// TIA Portal project "progettoPAGANOVOLZONE" (V17)
// Vorlageprojekt für das Buch mit Zielsystem S7-1200

(* hardware
DEVICE "S7-1200-Station_1"  S7-1200 Station
   slot 0: "Baugruppenträger_0"  Rack  V1.0
   slot 1: "PLC_1"  CPU 1215C DC/DC/DC  6ES7 215-1AG40-0XB0  V4.5
   slot 2: "DQ 2x24VDC _1"  SM 1222 DQ8 x 24VDC  6ES7 222-1BF30-0XB0  V1.0
DEVICE "HMI_1"  KTP900 Basic PN
   slot 0: "HMI_1"  KTP900 Basic PN  6AV2 123-2JB03-0AX0  17.0.0.0
   slot 1: "HMI_RT_1"  KTP900 Basic PN  6AV2 123-2JB03-0AX0  17.0.0.0
   slot 5: "HMI_1.IE_CP_1"  PROFINET Interface  17.0.0.0
      slot 1: "PROFINET Interface_1"  PROFINET Interface
         slot 1: "Port_1"  Port
*)

// ===== PLC "PLC_1"  CPU 1215C DC/DC/DC =====

VAR_GLOBAL   // PLC tag table "Standard-Variablentabelle"
   "Tag_1" AT %A0.0 : Bool;
   "Tag_2" AT %E0.0 : Bool;
   "Tag_3" AT %E0.1 : Bool;
   "Tag_4" AT %Q0.1 : Bool;
   "Tag_5" AT %I0.2 : Bool;
   "Tag_6" AT %Q0.2 : Bool;
   "Tag_7" AT %I0.3 : Bool;
   "Tag_8" AT %Q0.3 : Bool;
   "Tag_9" AT %I0.4 : Bool;
   "Tag_10" AT %Q0.4 : Bool;
   "Tag_11" AT %I0.5 : Bool;
   "Tag_12" AT %I0.6 : Bool;
   "Tag_13" AT %I0.7 : Bool;
   "Tag_14" AT %I1.0 : Bool;
   "Tag_15" AT %Q0.5 : Bool;
   "Tag_16" AT %Q0.6 : Bool;
   "Tag_17" AT %Q0.7 : Bool;
   "Tag_18" AT %Q1.0 : Bool;
   "Tag_19" AT %Q1.1 : Bool;
   "Tag_20" AT %I1.1 : Bool;
   "Tag_21" AT %I1.2 : Bool;
   "Tag_22" AT %Q1.2 : Bool;
   "Tag_23" AT %Q1.3 : Bool;
   "Tag_24" AT %I1.6 : Bool;
   "Tag_25" AT %ID30 : Real;
   "Tag_26" AT %I1.3 : Bool;
   "Tag_27" AT %I1.5 : Bool;
   "Tag_28" AT %I1.7 : Bool;
   "Tag_29" AT %Q1.4 : Bool;
   "Tag_30" AT %Q1.5 : Bool;
   "Tag_31" AT %Q1.6 : Bool;
   "Tag_32" AT %Q1.7 : Bool;
   "Tag_33" AT %I1.4 : Bool;
   "tag1" AT %M1.0 : Bool;
   "pezzi_scartati" AT %MW0 : Int;
   "allarme" AT %Q2.0 : Bool;
   "Tag_34" AT %I2.1 : Bool;
   "Tag_35" AT %I2.0 : Bool;
   "Tag_36" AT %I2.2 : Bool;
   "Tag_37" AT %I2.3 : Bool;
END_VAR

DATA_BLOCK "nastro1"   // DB1
{ S7_Optimized_Access := 'TRUE' }
VERSION : 0.1
// stored: InstanceOfName nastro
"nastro"
BEGIN
END_DATA_BLOCK

DATA_BLOCK "nastro2"   // DB2
{ S7_Optimized_Access := 'TRUE' }
VERSION : 0.1
// stored: InstanceOfName nastro
"nastro"
BEGIN
END_DATA_BLOCK

DATA_BLOCK "nastro3"   // DB3
{ S7_Optimized_Access := 'TRUE' }
VERSION : 0.1
// stored: InstanceOfName nastro
"nastro"
BEGIN
END_DATA_BLOCK

DATA_BLOCK "robotCentrale"   // DB5
{ S7_Optimized_Access := 'TRUE' }
VERSION : 0.1
// stored: InstanceOfName robotSD
"robotSD"
BEGIN
END_DATA_BLOCK

DATA_BLOCK "elevator1"   // DB7
{ S7_Optimized_Access := 'TRUE' }
VERSION : 0.1
// stored: InstanceOfName elevator
"elevator"
BEGIN
END_DATA_BLOCK

DATA_BLOCK "nastroCentrale1"   // DB8
{ S7_Optimized_Access := 'TRUE' }
VERSION : 0.1
// stored: InstanceOfName nastroCentrale
"nastroCentrale"
BEGIN
END_DATA_BLOCK

DATA_BLOCK "weight1"   // DB9
{ S7_Optimized_Access := 'TRUE' }
VERSION : 0.1
// stored: InstanceOfName weight
"weight"
BEGIN
END_DATA_BLOCK

DATA_BLOCK "NastroDirezionale1"   // DB10
{ S7_Optimized_Access := 'TRUE' }
VERSION : 0.1
// stored: InstanceOfName NastroDirezionale
"NastroDirezionale"
BEGIN
END_DATA_BLOCK

FUNCTION_BLOCK "robotSD"   // FB1, LAD
{ S7_Optimized_Access := 'TRUE' }
VERSION : 0.1
   VAR_INPUT
      workD : Bool;   // work del nastro destro
      workS : Bool;   // work del nastro sinistro
      grabsens : Bool;
      godownsens : Bool;
      movesens : Bool;
      rotateSens : Bool;
      occupato : Bool;   // sensore sul nastro d'arrivo
      tempot2 : Time := T#1s;
   END_VAR
   VAR_OUTPUT
      godown : Bool;
      grab : Bool;
      move : Bool;
      sinistra : Bool;
      destra : Bool;
      work_finishedD : Bool;
      work_finishedS : Bool;
   END_VAR
   VAR
      f0 : Bool;   // base
      "f1.1" : Bool;
      "f1.2" : Bool;
      f2 : Bool;
      f3 : Bool;
      f4 : Bool;
      "f5.1" : Bool;
      "f5.2" : Bool;
      f6 : Bool;
      f7 : Bool;
      f8 : Bool;
      f9 : Bool;
      "f9.1" : Bool;
      f10 : Bool;
      iniz : Bool;
      F_sensD : F_TRIG;   // falling del sensore destro
      F_sensS : F_TRIG;   // falling del sensore sinistro
      R_grabsens : R_TRIG;
      R_occupato : R_TRIG;
      F_godownsens : F_TRIG;
      F_movesens : F_TRIG;
      F_rotateSens : F_TRIG;   // falling del sensore di rotazione
      timer_f2 : TON_TIME;
      varDestra : Bool;
   END_VAR
   VAR_TEMP
      tr1 : Bool;   // sensore destro o sinistro falling edge
      tr2 : Bool;
      tr3 : Bool;
      tr4 : Bool;
      tr5 : Bool;
      tr6 : Bool;
      tr7 : Bool;
      tr8 : Bool;
      tr9 : Bool;
      tr10 : Bool;
      tr11 : Bool;
      tr12 : Bool;
      tr13 : Bool;
      tr14 : Bool;
      "tr14.1" : Bool;
      tr15 : Bool;
   END_VAR
   VAR_TEMP   // added for the SCL form of the ladder/FBD networks
      _w1 : Bool;
   END_VAR
BEGIN

REGION Network 1: inizializzazione
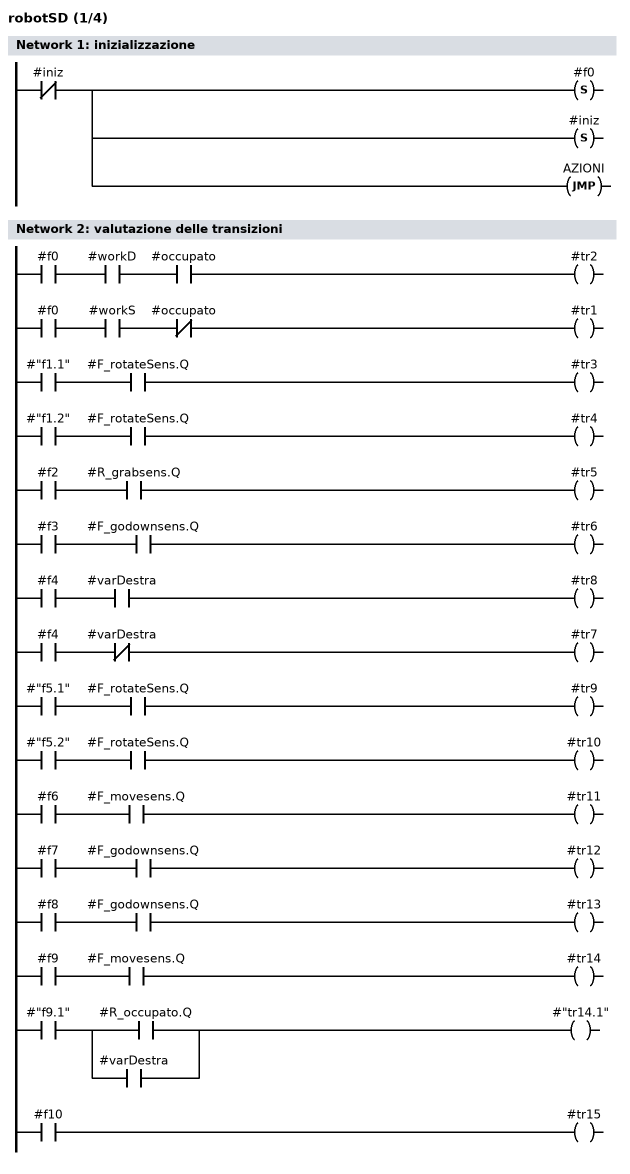
   RUNG wire#powerrail
      I_Contact( #iniz )
      wire#w1
      S_Coil( #f0 )
   END_RUNG
   RUNG wire#w1
      S_Coil( #iniz )
   END_RUNG
   RUNG wire#w1
      JumpCoil( AZIONI )
   END_RUNG
   // the same network as SCL:
   IF NOT #iniz THEN #f0 := TRUE; END_IF;
   #_w1 := NOT #iniz;
   IF #_w1 THEN
       #iniz := TRUE;
       GOTO AZIONI;
   END_IF;
END_REGION

REGION Network 2: valutazione delle transizioni
   RUNG wire#powerrail
      Contact( #f0 )
      Contact( #workD )
      Contact( #occupato )
      Coil( #tr2 )
   END_RUNG
   RUNG wire#powerrail
      Contact( #f0 )
      Contact( #workS )
      I_Contact( #occupato )
      Coil( #tr1 )
   END_RUNG
   RUNG wire#powerrail
      Contact( #"f1.1" )
      Contact( #F_rotateSens.Q )
      Coil( #tr3 )
   END_RUNG
   RUNG wire#powerrail
      Contact( #"f1.2" )
      Contact( #F_rotateSens.Q )
      Coil( #tr4 )
   END_RUNG
   RUNG wire#powerrail
      Contact( #f2 )
      Contact( #R_grabsens.Q )
      Coil( #tr5 )
   END_RUNG
   RUNG wire#powerrail
      Contact( #f3 )
      Contact( #F_godownsens.Q )
      Coil( #tr6 )
   END_RUNG
   RUNG wire#powerrail
      Contact( #f4 )
      Contact( #varDestra )
      Coil( #tr8 )
   END_RUNG
   RUNG wire#powerrail
      Contact( #f4 )
      I_Contact( #varDestra )
      Coil( #tr7 )
   END_RUNG
   RUNG wire#powerrail
      Contact( #"f5.1" )
      Contact( #F_rotateSens.Q )
      Coil( #tr9 )
   END_RUNG
   RUNG wire#powerrail
      Contact( #"f5.2" )
      Contact( #F_rotateSens.Q )
      Coil( #tr10 )
   END_RUNG
   RUNG wire#powerrail
      Contact( #f6 )
      Contact( #F_movesens.Q )
      Coil( #tr11 )
   END_RUNG
   RUNG wire#powerrail
      Contact( #f7 )
      Contact( #F_godownsens.Q )
      Coil( #tr12 )
   END_RUNG
   RUNG wire#powerrail
      Contact( #f8 )
      Contact( #F_godownsens.Q )
      Coil( #tr13 )
   END_RUNG
   RUNG wire#powerrail
      Contact( #f9 )
      Contact( #F_movesens.Q )
      Coil( #tr14 )
   END_RUNG
   RUNG wire#powerrail
      Contact( #"f9.1" )
      wire#w1
      Contact( #R_occupato.Q )
      wire#w2
      Coil( #"tr14.1" )
   END_RUNG
   RUNG wire#w1
      Contact( #varDestra )
   END_RUNG wire#w2
   RUNG wire#powerrail
      Contact( #f10 )
      Coil( #tr15 )
   END_RUNG
   // the same network as SCL:
   #tr2 := #f0 AND #workD AND #occupato;
   #tr1 := #f0 AND #workS AND NOT #occupato;
   #tr3 := #"f1.1" AND #F_rotateSens.Q;
   #tr4 := #"f1.2" AND #F_rotateSens.Q;
   #tr5 := #f2 AND #R_grabsens.Q;
   #tr6 := #f3 AND #F_godownsens.Q;
   #tr8 := #f4 AND #varDestra;
   #tr7 := #f4 AND NOT #varDestra;
   #tr9 := #"f5.1" AND #F_rotateSens.Q;
   #tr10 := #"f5.2" AND #F_rotateSens.Q;
   #tr11 := #f6 AND #F_movesens.Q;
   #tr12 := #f7 AND #F_godownsens.Q;
   #tr13 := #f8 AND #F_godownsens.Q;
   #tr14 := #f9 AND #F_movesens.Q;
   #"tr14.1" := #"f9.1" AND (#R_occupato.Q OR #varDestra);
   #tr15 := #f10;
END_REGION

REGION Network 3: aggiornamento della condizione
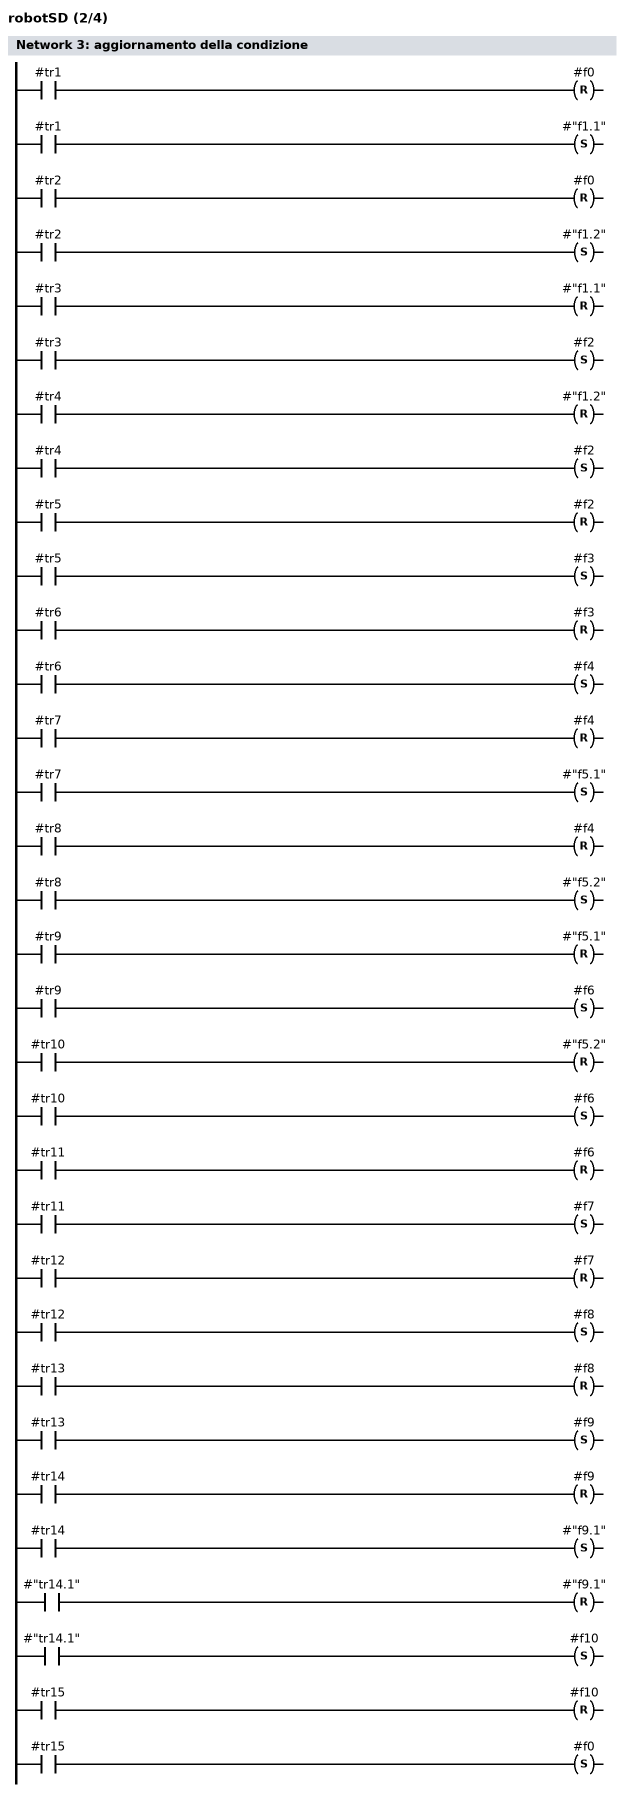
   RUNG wire#powerrail
      Contact( #tr1 )
      R_Coil( #f0 )
   END_RUNG
   RUNG wire#powerrail
      Contact( #tr1 )
      S_Coil( #"f1.1" )
   END_RUNG
   RUNG wire#powerrail
      Contact( #tr2 )
      R_Coil( #f0 )
   END_RUNG
   RUNG wire#powerrail
      Contact( #tr2 )
      S_Coil( #"f1.2" )
   END_RUNG
   RUNG wire#powerrail
      Contact( #tr3 )
      R_Coil( #"f1.1" )
   END_RUNG
   RUNG wire#powerrail
      Contact( #tr3 )
      S_Coil( #f2 )
   END_RUNG
   RUNG wire#powerrail
      Contact( #tr4 )
      R_Coil( #"f1.2" )
   END_RUNG
   RUNG wire#powerrail
      Contact( #tr4 )
      S_Coil( #f2 )
   END_RUNG
   RUNG wire#powerrail
      Contact( #tr5 )
      R_Coil( #f2 )
   END_RUNG
   RUNG wire#powerrail
      Contact( #tr5 )
      S_Coil( #f3 )
   END_RUNG
   RUNG wire#powerrail
      Contact( #tr6 )
      R_Coil( #f3 )
   END_RUNG
   RUNG wire#powerrail
      Contact( #tr6 )
      S_Coil( #f4 )
   END_RUNG
   RUNG wire#powerrail
      Contact( #tr7 )
      R_Coil( #f4 )
   END_RUNG
   RUNG wire#powerrail
      Contact( #tr7 )
      S_Coil( #"f5.1" )
   END_RUNG
   RUNG wire#powerrail
      Contact( #tr8 )
      R_Coil( #f4 )
   END_RUNG
   RUNG wire#powerrail
      Contact( #tr8 )
      S_Coil( #"f5.2" )
   END_RUNG
   RUNG wire#powerrail
      Contact( #tr9 )
      R_Coil( #"f5.1" )
   END_RUNG
   RUNG wire#powerrail
      Contact( #tr9 )
      S_Coil( #f6 )
   END_RUNG
   RUNG wire#powerrail
      Contact( #tr10 )
      R_Coil( #"f5.2" )
   END_RUNG
   RUNG wire#powerrail
      Contact( #tr10 )
      S_Coil( #f6 )
   END_RUNG
   RUNG wire#powerrail
      Contact( #tr11 )
      R_Coil( #f6 )
   END_RUNG
   RUNG wire#powerrail
      Contact( #tr11 )
      S_Coil( #f7 )
   END_RUNG
   RUNG wire#powerrail
      Contact( #tr12 )
      R_Coil( #f7 )
   END_RUNG
   RUNG wire#powerrail
      Contact( #tr12 )
      S_Coil( #f8 )
   END_RUNG
   RUNG wire#powerrail
      Contact( #tr13 )
      R_Coil( #f8 )
   END_RUNG
   RUNG wire#powerrail
      Contact( #tr13 )
      S_Coil( #f9 )
   END_RUNG
   RUNG wire#powerrail
      Contact( #tr14 )
      R_Coil( #f9 )
   END_RUNG
   RUNG wire#powerrail
      Contact( #tr14 )
      S_Coil( #"f9.1" )
   END_RUNG
   RUNG wire#powerrail
      Contact( #"tr14.1" )
      R_Coil( #"f9.1" )
   END_RUNG
   RUNG wire#powerrail
      Contact( #"tr14.1" )
      S_Coil( #f10 )
   END_RUNG
   RUNG wire#powerrail
      Contact( #tr15 )
      R_Coil( #f10 )
   END_RUNG
   RUNG wire#powerrail
      Contact( #tr15 )
      S_Coil( #f0 )
   END_RUNG
   // the same network as SCL:
   IF #tr1 THEN
       #f0 := FALSE;
       #"f1.1" := TRUE;
   END_IF;
   IF #tr2 THEN
       #f0 := FALSE;
       #"f1.2" := TRUE;
   END_IF;
   IF #tr3 THEN
       #"f1.1" := FALSE;
       #f2 := TRUE;
   END_IF;
   IF #tr4 THEN
       #"f1.2" := FALSE;
       #f2 := TRUE;
   END_IF;
   IF #tr5 THEN
       #f2 := FALSE;
       #f3 := TRUE;
   END_IF;
   IF #tr6 THEN
       #f3 := FALSE;
       #f4 := TRUE;
   END_IF;
   IF #tr7 THEN
       #f4 := FALSE;
       #"f5.1" := TRUE;
   END_IF;
   IF #tr8 THEN
       #f4 := FALSE;
       #"f5.2" := TRUE;
   END_IF;
   IF #tr9 THEN
       #"f5.1" := FALSE;
       #f6 := TRUE;
   END_IF;
   IF #tr10 THEN
       #"f5.2" := FALSE;
       #f6 := TRUE;
   END_IF;
   IF #tr11 THEN
       #f6 := FALSE;
       #f7 := TRUE;
   END_IF;
   IF #tr12 THEN
       #f7 := FALSE;
       #f8 := TRUE;
   END_IF;
   IF #tr13 THEN
       #f8 := FALSE;
       #f9 := TRUE;
   END_IF;
   IF #tr14 THEN
       #f9 := FALSE;
       #"f9.1" := TRUE;
   END_IF;
   IF #"tr14.1" THEN
       #"f9.1" := FALSE;
       #f10 := TRUE;
   END_IF;
   IF #tr15 THEN
       #f10 := FALSE;
       #f0 := TRUE;
   END_IF;
END_REGION

REGION Network 4: esecuzione delle azioni
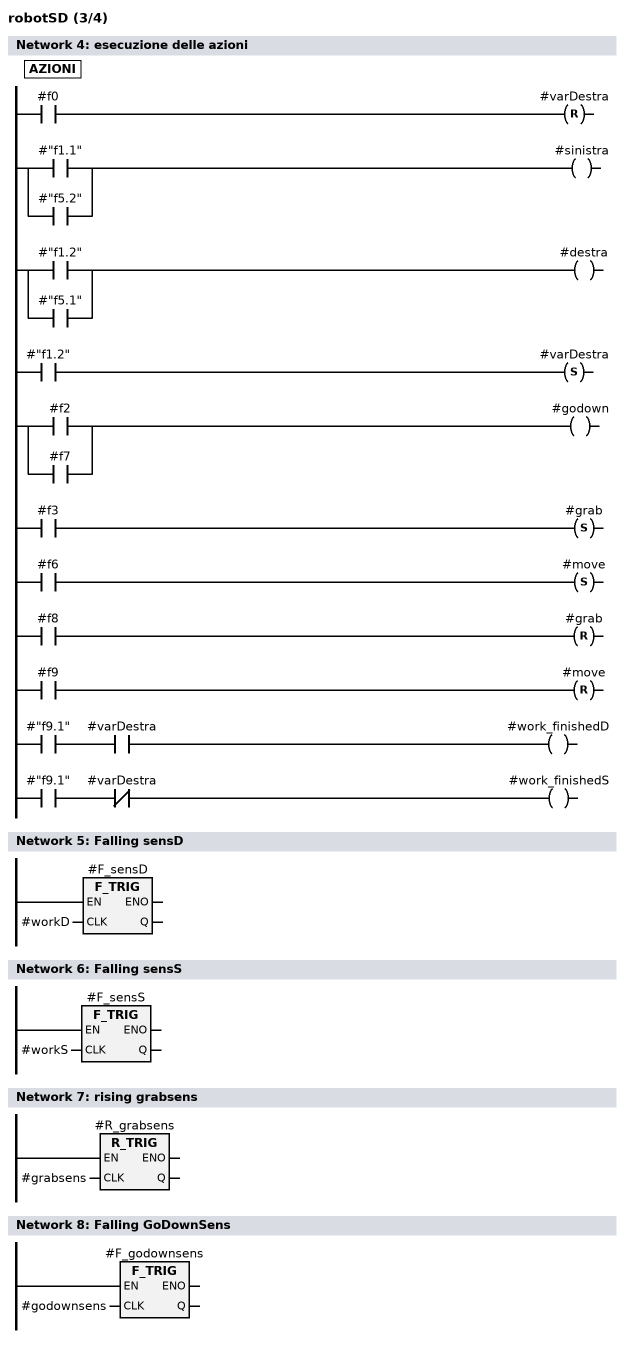
   Label( AZIONI )
   RUNG wire#powerrail
      Contact( #f0 )
      R_Coil( #varDestra )
   END_RUNG
   RUNG wire#powerrail
      Contact( #"f1.1" )
      wire#w1
      Coil( #sinistra )
   END_RUNG
   RUNG wire#powerrail
      Contact( #"f5.2" )
   END_RUNG wire#w1
   RUNG wire#powerrail
      Contact( #"f1.2" )
      wire#w2
      Coil( #destra )
   END_RUNG
   RUNG wire#powerrail
      Contact( #"f5.1" )
   END_RUNG wire#w2
   RUNG wire#powerrail
      Contact( #"f1.2" )
      S_Coil( #varDestra )
   END_RUNG
   RUNG wire#powerrail
      Contact( #f2 )
      wire#w3
      Coil( #godown )
   END_RUNG
   RUNG wire#powerrail
      Contact( #f7 )
   END_RUNG wire#w3
   RUNG wire#powerrail
      Contact( #f3 )
      S_Coil( #grab )
   END_RUNG
   RUNG wire#powerrail
      Contact( #f6 )
      S_Coil( #move )
   END_RUNG
   RUNG wire#powerrail
      Contact( #f8 )
      R_Coil( #grab )
   END_RUNG
   RUNG wire#powerrail
      Contact( #f9 )
      R_Coil( #move )
   END_RUNG
   RUNG wire#powerrail
      Contact( #"f9.1" )
      Contact( #varDestra )
      Coil( #work_finishedD )
   END_RUNG
   RUNG wire#powerrail
      Contact( #"f9.1" )
      I_Contact( #varDestra )
      Coil( #work_finishedS )
   END_RUNG
   // the same network as SCL:
   AZIONI:
   IF #f0 THEN #varDestra := FALSE; END_IF;
   #sinistra := #"f1.1" OR #"f5.2";
   #destra := #"f1.2" OR #"f5.1";
   IF #"f1.2" THEN #varDestra := TRUE; END_IF;
   #godown := #f2 OR #f7;
   IF #f3 THEN #grab := TRUE; END_IF;
   IF #f6 THEN #move := TRUE; END_IF;
   IF #f8 THEN #grab := FALSE; END_IF;
   IF #f9 THEN #move := FALSE; END_IF;
   #work_finishedD := #"f9.1" AND #varDestra;
   #work_finishedS := #"f9.1" AND NOT #varDestra;
END_REGION

REGION Network 5: Falling sensD
   #F_sensD(CLK := #workD);   // F_TRIG
END_REGION

REGION Network 6: Falling sensS
   #F_sensS(CLK := #workS);   // F_TRIG
END_REGION

REGION Network 7: rising grabsens
   #R_grabsens(CLK := #grabsens);   // R_TRIG
END_REGION

REGION Network 8: Falling GoDownSens
   #F_godownsens(CLK := #godownsens);   // F_TRIG
END_REGION

REGION Network 9: Falling MoveSens
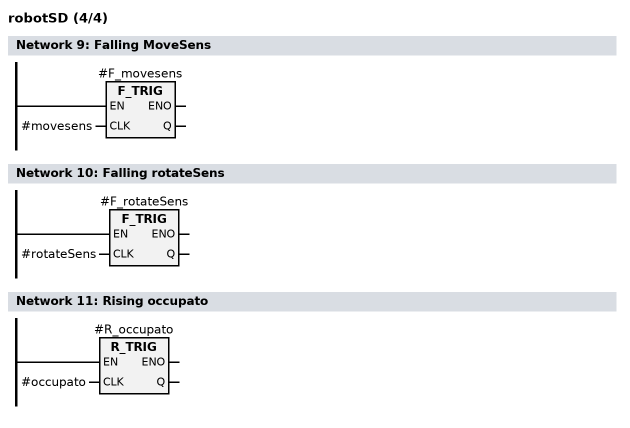
   #F_movesens(CLK := #movesens);   // F_TRIG
END_REGION

REGION Network 10: Falling rotateSens
   #F_rotateSens(CLK := #rotateSens);   // F_TRIG
END_REGION

REGION Network 11: Rising occupato
   #R_occupato(CLK := #occupato);   // R_TRIG
END_REGION
END_FUNCTION_BLOCK

FUNCTION_BLOCK "nastro"   // FB2, LAD
{ S7_Optimized_Access := 'TRUE' }
VERSION : 0.1
   VAR_INPUT
      s : Bool;
      work_finished : Bool;
   END_VAR
   VAR_OUTPUT
      motor : Bool;
      work : Bool;
   END_VAR
   VAR
      f0 : Bool;
      f1 : Bool;
      f2 : Bool;
      init : Bool;
      F_S : F_TRIG;
      F_Finished : F_TRIG;
      R_S : R_TRIG;
   END_VAR
   VAR_TEMP
      tr1 : Bool;
      tr3 : Bool;
      tr2 : Bool;
   END_VAR
   VAR_TEMP   // added for the SCL form of the ladder/FBD networks
      _w1 : Bool;
   END_VAR
BEGIN

REGION Network 1: inizializzazione
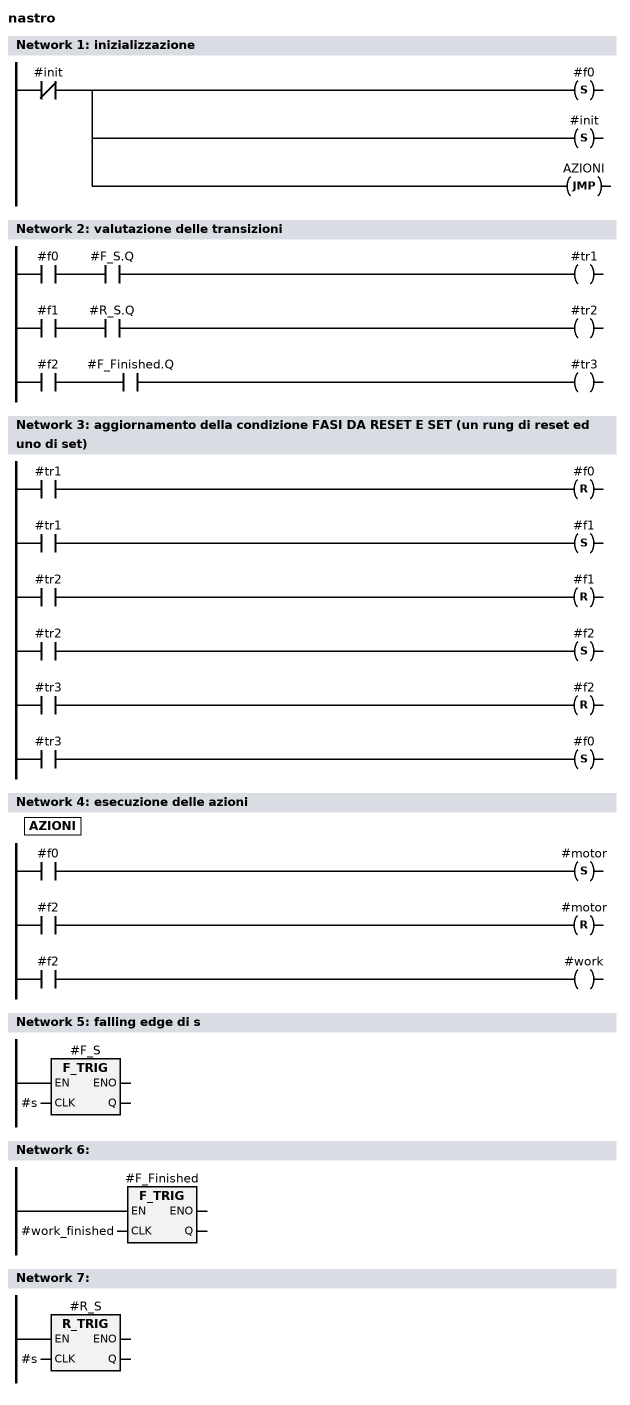
   RUNG wire#powerrail
      I_Contact( #init )
      wire#w1
      S_Coil( #f0 )
   END_RUNG
   RUNG wire#w1
      S_Coil( #init )
   END_RUNG
   RUNG wire#w1
      JumpCoil( AZIONI )
   END_RUNG
   // the same network as SCL:
   IF NOT #init THEN #f0 := TRUE; END_IF;
   #_w1 := NOT #init;
   IF #_w1 THEN
       #init := TRUE;
       GOTO AZIONI;
   END_IF;
END_REGION

REGION Network 2: valutazione delle transizioni
   RUNG wire#powerrail
      Contact( #f0 )
      Contact( #F_S.Q )
      Coil( #tr1 )
   END_RUNG
   RUNG wire#powerrail
      Contact( #f1 )
      Contact( #R_S.Q )
      Coil( #tr2 )
   END_RUNG
   RUNG wire#powerrail
      Contact( #f2 )
      Contact( #F_Finished.Q )
      Coil( #tr3 )
   END_RUNG
   // the same network as SCL:
   #tr1 := #f0 AND #F_S.Q;
   #tr2 := #f1 AND #R_S.Q;
   #tr3 := #f2 AND #F_Finished.Q;
END_REGION

REGION Network 3: aggiornamento della condizione FASI DA RESET E SET (un rung di reset ed uno di set)
   RUNG wire#powerrail
      Contact( #tr1 )
      R_Coil( #f0 )
   END_RUNG
   RUNG wire#powerrail
      Contact( #tr1 )
      S_Coil( #f1 )
   END_RUNG
   RUNG wire#powerrail
      Contact( #tr2 )
      R_Coil( #f1 )
   END_RUNG
   RUNG wire#powerrail
      Contact( #tr2 )
      S_Coil( #f2 )
   END_RUNG
   RUNG wire#powerrail
      Contact( #tr3 )
      R_Coil( #f2 )
   END_RUNG
   RUNG wire#powerrail
      Contact( #tr3 )
      S_Coil( #f0 )
   END_RUNG
   // the same network as SCL:
   IF #tr1 THEN
       #f0 := FALSE;
       #f1 := TRUE;
   END_IF;
   IF #tr2 THEN
       #f1 := FALSE;
       #f2 := TRUE;
   END_IF;
   IF #tr3 THEN
       #f2 := FALSE;
       #f0 := TRUE;
   END_IF;
END_REGION

REGION Network 4: esecuzione delle azioni
   Label( AZIONI )
   RUNG wire#powerrail
      Contact( #f0 )
      S_Coil( #motor )
   END_RUNG
   RUNG wire#powerrail
      Contact( #f2 )
      R_Coil( #motor )
   END_RUNG
   RUNG wire#powerrail
      Contact( #f2 )
      Coil( #work )
   END_RUNG
   // the same network as SCL:
   AZIONI:
   IF #f0 THEN #motor := TRUE; END_IF;
   IF #f2 THEN #motor := FALSE; END_IF;
   #work := #f2;
END_REGION

REGION Network 5: falling edge di s
   #F_S(CLK := #s);   // F_TRIG
END_REGION

REGION Network 6
   #F_Finished(CLK := #work_finished);   // F_TRIG
END_REGION

REGION Network 7
   #R_S(CLK := #s);   // R_TRIG
END_REGION
END_FUNCTION_BLOCK

FUNCTION_BLOCK "elevator"   // FB3, LAD
TITLE = elevatore
{ S7_Optimized_Access := 'TRUE' }
VERSION : 0.1
   VAR_INPUT
      piano : Bool;
      sensDXup : Bool;
      boxon : Bool;
      sensSTOP : Bool;
      elevatorDown : Bool;
      sensDXdown : Bool;
      sensS : Bool;
   END_VAR
   VAR_OUTPUT
      down : Bool;
      AVA : Bool;
      up : Bool;
      work_finished : Bool;
   END_VAR
   VAR
      f0 : Bool;   // work finished
      "f0.1" : Bool;
      "f1.1" : Bool;   // piano 1
      "f1.2" : Bool;   // piano 0
      "f2.1" : Bool;   // sopra
      "f3.1" : Bool;   // piano 1, scendere fino a piano 0
      f4 : Bool;
      init : Bool;
      F_sensDXup : F_TRIG;
      F_boxOn : F_TRIG;
      F_sensDXdown : F_TRIG;
      F_sensS : F_TRIG;
      R_sensStop : R_TRIG;
      R_elevatorDown : R_TRIG;
   END_VAR
   VAR_TEMP
      tr1 : Bool;
      tr2 : Bool;
      tr3 : Bool;
      "tr3.1" : Bool;
      tr4 : Bool;
      tr5 : Bool;
      tr6 : Bool;
      tr7 : Bool;
      "tr0.1" : Bool;
   END_VAR
   VAR_TEMP   // added for the SCL form of the ladder/FBD networks
      _w1 : Bool;
   END_VAR
BEGIN

REGION Network 1: inizializzazione
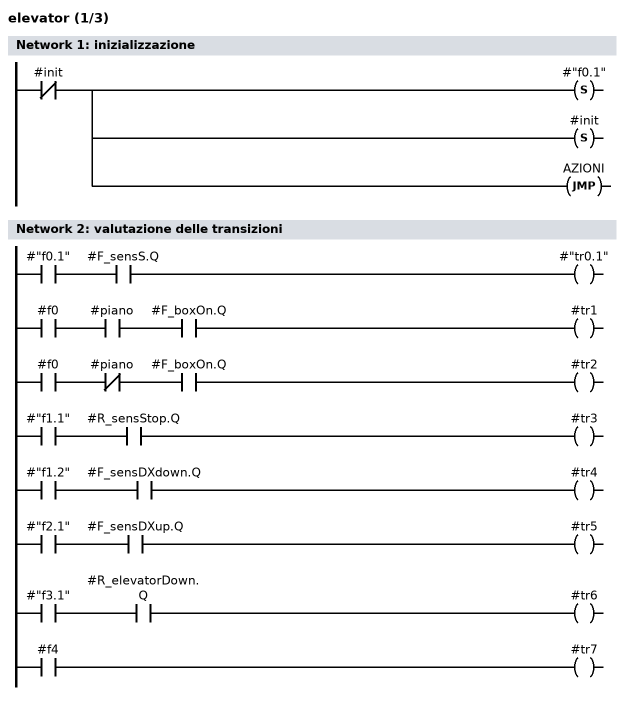
   RUNG wire#powerrail
      I_Contact( #init )
      wire#w1
      S_Coil( #"f0.1" )
   END_RUNG
   RUNG wire#w1
      S_Coil( #init )
   END_RUNG
   RUNG wire#w1
      JumpCoil( AZIONI )
   END_RUNG
   // the same network as SCL:
   IF NOT #init THEN #"f0.1" := TRUE; END_IF;
   #_w1 := NOT #init;
   IF #_w1 THEN
       #init := TRUE;
       GOTO AZIONI;
   END_IF;
END_REGION

REGION Network 2: valutazione delle transizioni
   RUNG wire#powerrail
      Contact( #"f0.1" )
      Contact( #F_sensS.Q )
      Coil( #"tr0.1" )
   END_RUNG
   RUNG wire#powerrail
      Contact( #f0 )
      Contact( #piano )
      Contact( #F_boxOn.Q )
      Coil( #tr1 )
   END_RUNG
   RUNG wire#powerrail
      Contact( #f0 )
      I_Contact( #piano )
      Contact( #F_boxOn.Q )
      Coil( #tr2 )
   END_RUNG
   RUNG wire#powerrail
      Contact( #"f1.1" )
      Contact( #R_sensStop.Q )
      Coil( #tr3 )
   END_RUNG
   RUNG wire#powerrail
      Contact( #"f1.2" )
      Contact( #F_sensDXdown.Q )
      Coil( #tr4 )
   END_RUNG
   RUNG wire#powerrail
      Contact( #"f2.1" )
      Contact( #F_sensDXup.Q )
      Coil( #tr5 )
   END_RUNG
   RUNG wire#powerrail
      Contact( #"f3.1" )
      Contact( #R_elevatorDown.Q )
      Coil( #tr6 )
   END_RUNG
   RUNG wire#powerrail
      Contact( #f4 )
      Coil( #tr7 )
   END_RUNG
   // the same network as SCL:
   #"tr0.1" := #"f0.1" AND #F_sensS.Q;
   #tr1 := #f0 AND #piano AND #F_boxOn.Q;
   #tr2 := #f0 AND NOT #piano AND #F_boxOn.Q;
   #tr3 := #"f1.1" AND #R_sensStop.Q;
   #tr4 := #"f1.2" AND #F_sensDXdown.Q;
   #tr5 := #"f2.1" AND #F_sensDXup.Q;
   #tr6 := #"f3.1" AND #R_elevatorDown.Q;
   #tr7 := #f4;
END_REGION

REGION Network 3: work finished
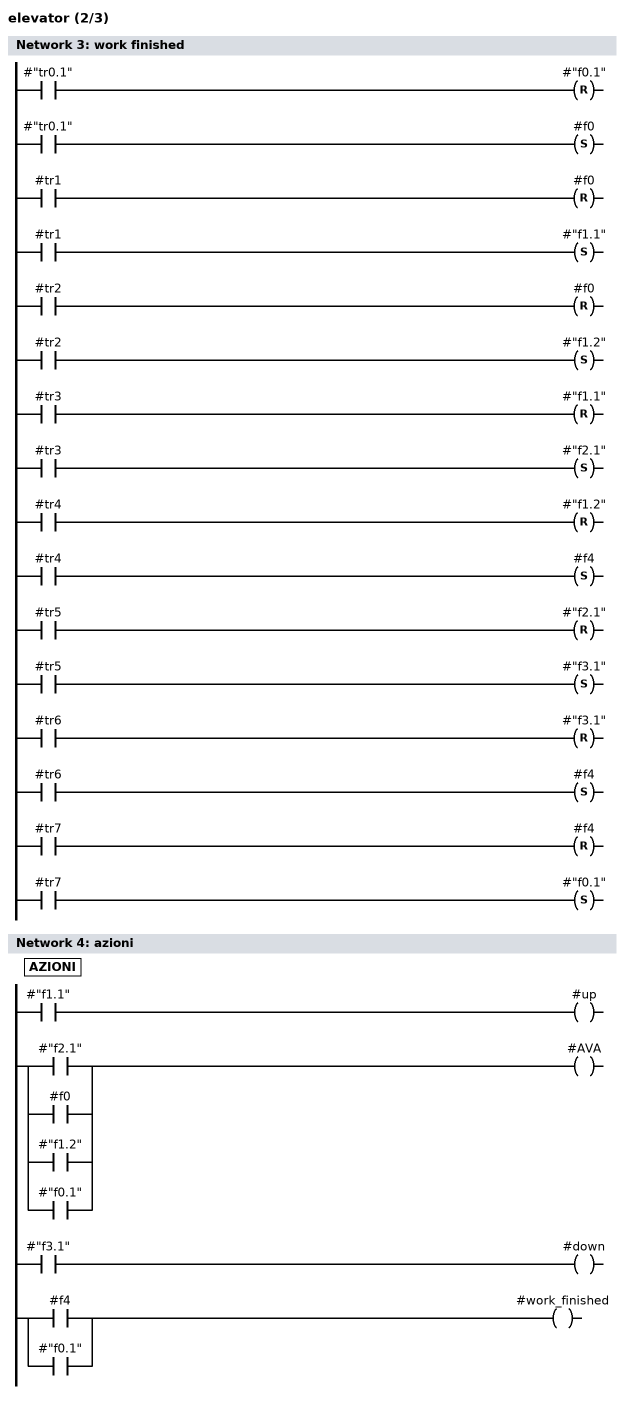
   RUNG wire#powerrail
      Contact( #"tr0.1" )
      R_Coil( #"f0.1" )
   END_RUNG
   RUNG wire#powerrail
      Contact( #"tr0.1" )
      S_Coil( #f0 )
   END_RUNG
   RUNG wire#powerrail
      Contact( #tr1 )
      R_Coil( #f0 )
   END_RUNG
   RUNG wire#powerrail
      Contact( #tr1 )
      S_Coil( #"f1.1" )
   END_RUNG
   RUNG wire#powerrail
      Contact( #tr2 )
      R_Coil( #f0 )
   END_RUNG
   RUNG wire#powerrail
      Contact( #tr2 )
      S_Coil( #"f1.2" )
   END_RUNG
   RUNG wire#powerrail
      Contact( #tr3 )
      R_Coil( #"f1.1" )
   END_RUNG
   RUNG wire#powerrail
      Contact( #tr3 )
      S_Coil( #"f2.1" )
   END_RUNG
   RUNG wire#powerrail
      Contact( #tr4 )
      R_Coil( #"f1.2" )
   END_RUNG
   RUNG wire#powerrail
      Contact( #tr4 )
      S_Coil( #f4 )
   END_RUNG
   RUNG wire#powerrail
      Contact( #tr5 )
      R_Coil( #"f2.1" )
   END_RUNG
   RUNG wire#powerrail
      Contact( #tr5 )
      S_Coil( #"f3.1" )
   END_RUNG
   RUNG wire#powerrail
      Contact( #tr6 )
      R_Coil( #"f3.1" )
   END_RUNG
   RUNG wire#powerrail
      Contact( #tr6 )
      S_Coil( #f4 )
   END_RUNG
   RUNG wire#powerrail
      Contact( #tr7 )
      R_Coil( #f4 )
   END_RUNG
   RUNG wire#powerrail
      Contact( #tr7 )
      S_Coil( #"f0.1" )
   END_RUNG
   // the same network as SCL:
   IF #"tr0.1" THEN
       #"f0.1" := FALSE;
       #f0 := TRUE;
   END_IF;
   IF #tr1 THEN
       #f0 := FALSE;
       #"f1.1" := TRUE;
   END_IF;
   IF #tr2 THEN
       #f0 := FALSE;
       #"f1.2" := TRUE;
   END_IF;
   IF #tr3 THEN
       #"f1.1" := FALSE;
       #"f2.1" := TRUE;
   END_IF;
   IF #tr4 THEN
       #"f1.2" := FALSE;
       #f4 := TRUE;
   END_IF;
   IF #tr5 THEN
       #"f2.1" := FALSE;
       #"f3.1" := TRUE;
   END_IF;
   IF #tr6 THEN
       #"f3.1" := FALSE;
       #f4 := TRUE;
   END_IF;
   IF #tr7 THEN
       #f4 := FALSE;
       #"f0.1" := TRUE;
   END_IF;
END_REGION

REGION Network 4: azioni
   Label( AZIONI )
   RUNG wire#powerrail
      Contact( #"f1.1" )
      Coil( #up )
   END_RUNG
   RUNG wire#powerrail
      Contact( #"f2.1" )
      wire#w1
      Coil( #AVA )
   END_RUNG
   RUNG wire#powerrail
      Contact( #f0 )
   END_RUNG wire#w1
   RUNG wire#powerrail
      Contact( #"f1.2" )
   END_RUNG wire#w1
   RUNG wire#powerrail
      Contact( #"f0.1" )
   END_RUNG wire#w1
   RUNG wire#powerrail
      Contact( #"f3.1" )
      Coil( #down )
   END_RUNG
   RUNG wire#powerrail
      Contact( #f4 )
      wire#w2
      Coil( #work_finished )
   END_RUNG
   RUNG wire#powerrail
      Contact( #"f0.1" )
   END_RUNG wire#w2
   // the same network as SCL:
   AZIONI:
   #up := #"f1.1";
   #AVA := #"f2.1" OR #f0 OR #"f1.2" OR #"f0.1";
   #down := #"f3.1";
   #work_finished := #f4 OR #"f0.1";
END_REGION

REGION Network 5
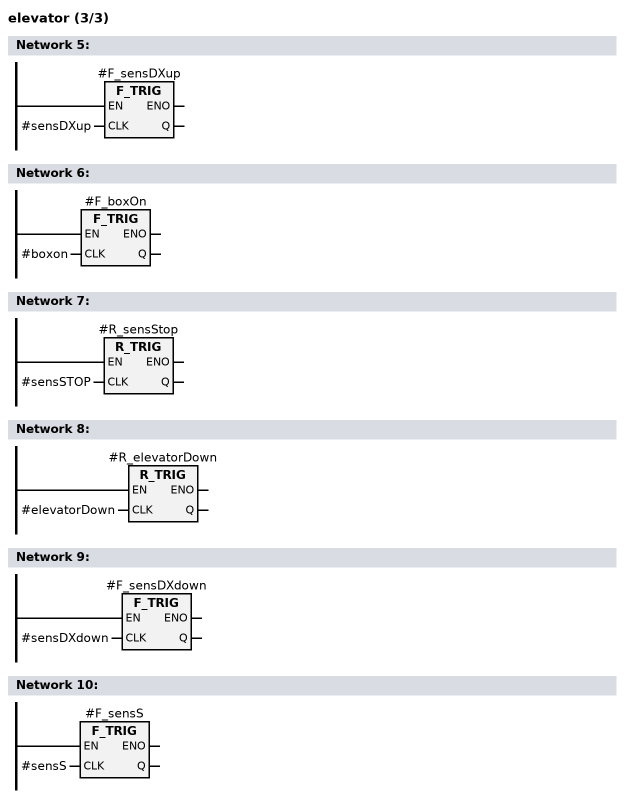
   #F_sensDXup(CLK := #sensDXup);   // F_TRIG
END_REGION

REGION Network 6
   #F_boxOn(CLK := #boxon);   // F_TRIG
END_REGION

REGION Network 7
   #R_sensStop(CLK := #sensSTOP);   // R_TRIG
END_REGION

REGION Network 8
   #R_elevatorDown(CLK := #elevatorDown);   // R_TRIG
END_REGION

REGION Network 9
   #F_sensDXdown(CLK := #sensDXdown);   // F_TRIG
END_REGION

REGION Network 10
   #F_sensS(CLK := #sensS);   // F_TRIG
END_REGION
END_FUNCTION_BLOCK

FUNCTION_BLOCK "weight"   // FB4, LAD
{ S7_Optimized_Access := 'TRUE' }
VERSION : 0.1
   VAR_INPUT
      weight : Real;
      tempot2 : Time := T#2s;
      occupato2 : Bool;
      prontoDopo : Bool;
   END_VAR
   VAR_OUTPUT
      piano : Bool;   // false=piano terra; true=primo piano
      workFinished : Bool;
      AVA : Bool;
   END_VAR
   VAR
      f0 : Bool;
      f1 : Bool;
      "f0.1" : Bool;
      "f2.1" : Bool;
      "f2.2" : Bool;
      f3 : Bool;
      iniz : Bool;
      "timer" : TON_TIME;
      F_occupato2 : F_TRIG;
   END_VAR
   VAR_TEMP
      tr1 : Bool;
      "tr0.1" : Bool;
      tr2 : Bool;
      tr3 : Bool;
      tr4 : Bool;
      tr5 : Bool;
   END_VAR
   VAR_TEMP   // added for the SCL form of the ladder/FBD networks
      _w1 : Bool;
   END_VAR
BEGIN

REGION Network 1: inizializzazione
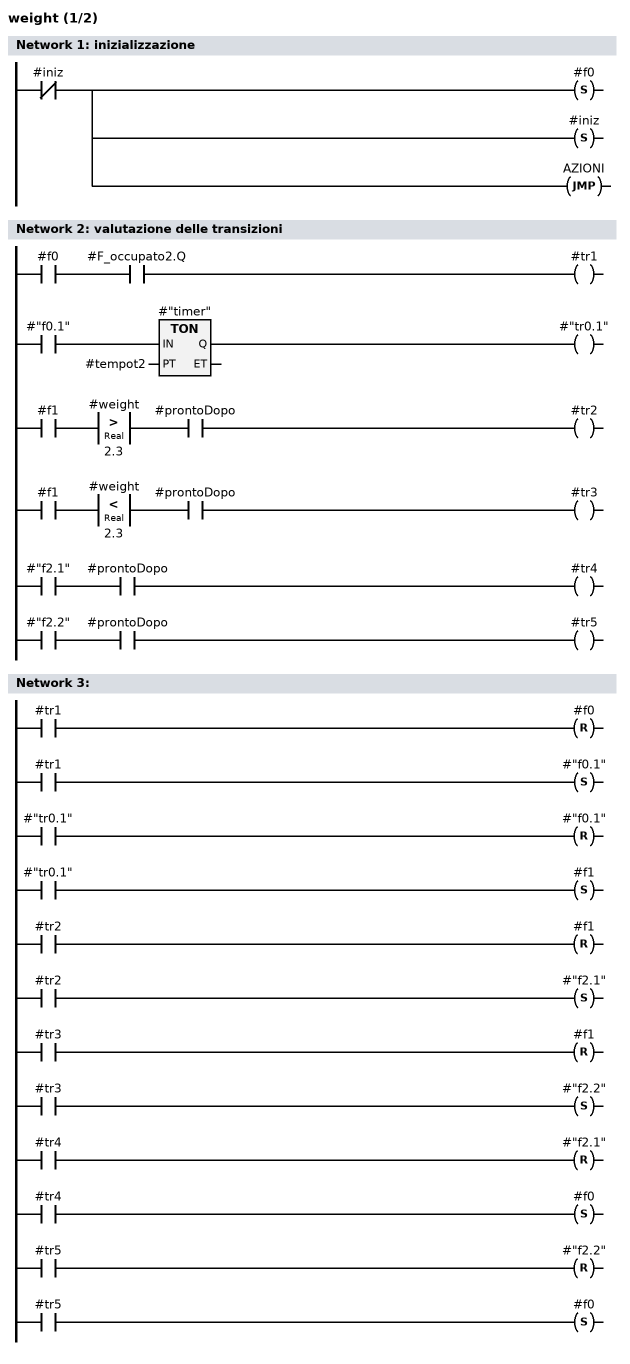
   RUNG wire#powerrail
      I_Contact( #iniz )
      wire#w1
      S_Coil( #f0 )
   END_RUNG
   RUNG wire#w1
      S_Coil( #iniz )
   END_RUNG
   RUNG wire#w1
      JumpCoil( AZIONI )
   END_RUNG
   // the same network as SCL:
   IF NOT #iniz THEN #f0 := TRUE; END_IF;
   #_w1 := NOT #iniz;
   IF #_w1 THEN
       #iniz := TRUE;
       GOTO AZIONI;
   END_IF;
END_REGION

REGION Network 2: valutazione delle transizioni
   #tr1 := #f0 AND #F_occupato2.Q;
   #"timer"(IN := #"f0.1", PT := #tempot2);   // TON
   #"tr0.1" := #"timer".Q;
   #tr2 := #f1 AND (#weight > 2.3) AND #prontoDopo;
   #tr3 := #f1 AND (#weight < 2.3) AND #prontoDopo;
   #tr4 := #"f2.1" AND #prontoDopo;
   #tr5 := #"f2.2" AND #prontoDopo;
END_REGION

REGION Network 3
   RUNG wire#powerrail
      Contact( #tr1 )
      R_Coil( #f0 )
   END_RUNG
   RUNG wire#powerrail
      Contact( #tr1 )
      S_Coil( #"f0.1" )
   END_RUNG
   RUNG wire#powerrail
      Contact( #"tr0.1" )
      R_Coil( #"f0.1" )
   END_RUNG
   RUNG wire#powerrail
      Contact( #"tr0.1" )
      S_Coil( #f1 )
   END_RUNG
   RUNG wire#powerrail
      Contact( #tr2 )
      R_Coil( #f1 )
   END_RUNG
   RUNG wire#powerrail
      Contact( #tr2 )
      S_Coil( #"f2.1" )
   END_RUNG
   RUNG wire#powerrail
      Contact( #tr3 )
      R_Coil( #f1 )
   END_RUNG
   RUNG wire#powerrail
      Contact( #tr3 )
      S_Coil( #"f2.2" )
   END_RUNG
   RUNG wire#powerrail
      Contact( #tr4 )
      R_Coil( #"f2.1" )
   END_RUNG
   RUNG wire#powerrail
      Contact( #tr4 )
      S_Coil( #f0 )
   END_RUNG
   RUNG wire#powerrail
      Contact( #tr5 )
      R_Coil( #"f2.2" )
   END_RUNG
   RUNG wire#powerrail
      Contact( #tr5 )
      S_Coil( #f0 )
   END_RUNG
   // the same network as SCL:
   IF #tr1 THEN
       #f0 := FALSE;
       #"f0.1" := TRUE;
   END_IF;
   IF #"tr0.1" THEN
       #"f0.1" := FALSE;
       #f1 := TRUE;
   END_IF;
   IF #tr2 THEN
       #f1 := FALSE;
       #"f2.1" := TRUE;
   END_IF;
   IF #tr3 THEN
       #f1 := FALSE;
       #"f2.2" := TRUE;
   END_IF;
   IF #tr4 THEN
       #"f2.1" := FALSE;
       #f0 := TRUE;
   END_IF;
   IF #tr5 THEN
       #"f2.2" := FALSE;
       #f0 := TRUE;
   END_IF;
END_REGION

REGION Network 4: azioni
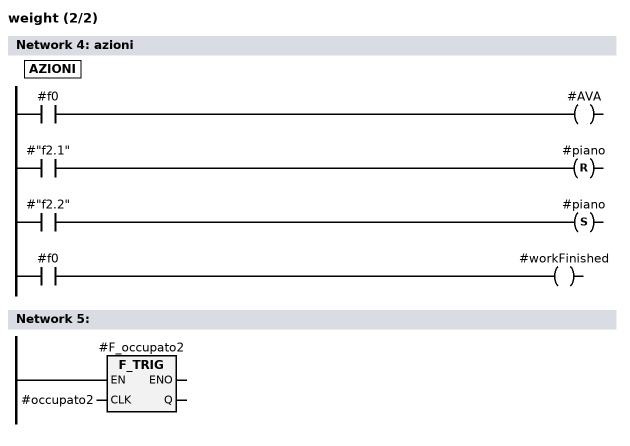
   Label( AZIONI )
   RUNG wire#powerrail
      Contact( #f0 )
      Coil( #AVA )
   END_RUNG
   RUNG wire#powerrail
      Contact( #"f2.1" )
      R_Coil( #piano )
   END_RUNG
   RUNG wire#powerrail
      Contact( #"f2.2" )
      S_Coil( #piano )
   END_RUNG
   RUNG wire#powerrail
      Contact( #f0 )
      Coil( #workFinished )
   END_RUNG
   // the same network as SCL:
   AZIONI:
   #AVA := #f0;
   IF #"f2.1" THEN #piano := FALSE; END_IF;
   IF #"f2.2" THEN #piano := TRUE; END_IF;
   #workFinished := #f0;
END_REGION

REGION Network 5
   #F_occupato2(CLK := #occupato2);   // F_TRIG
END_REGION
END_FUNCTION_BLOCK

FUNCTION_BLOCK "nastroCentrale"   // FB5, LAD
{ S7_Optimized_Access := 'TRUE' }
VERSION : 0.1
   VAR_INPUT
      work : Bool;   // work sinistro del robot centrale
      s : Bool;
      prontoDopo : Bool;
      sn : Bool;
   END_VAR
   VAR_OUTPUT
      motor : Bool;
   END_VAR
   VAR
      init : Bool;
      f0 : Bool;
      f1 : Bool;
      F_S : F_TRIG;
      F_SN : F_TRIG;
   END_VAR
   VAR_TEMP
      tr1 : Bool;
      tr2 : Bool;
   END_VAR
   VAR_TEMP   // added for the SCL form of the ladder/FBD networks
      _w1 : Bool;
   END_VAR
BEGIN

REGION Network 1: inizializzazione
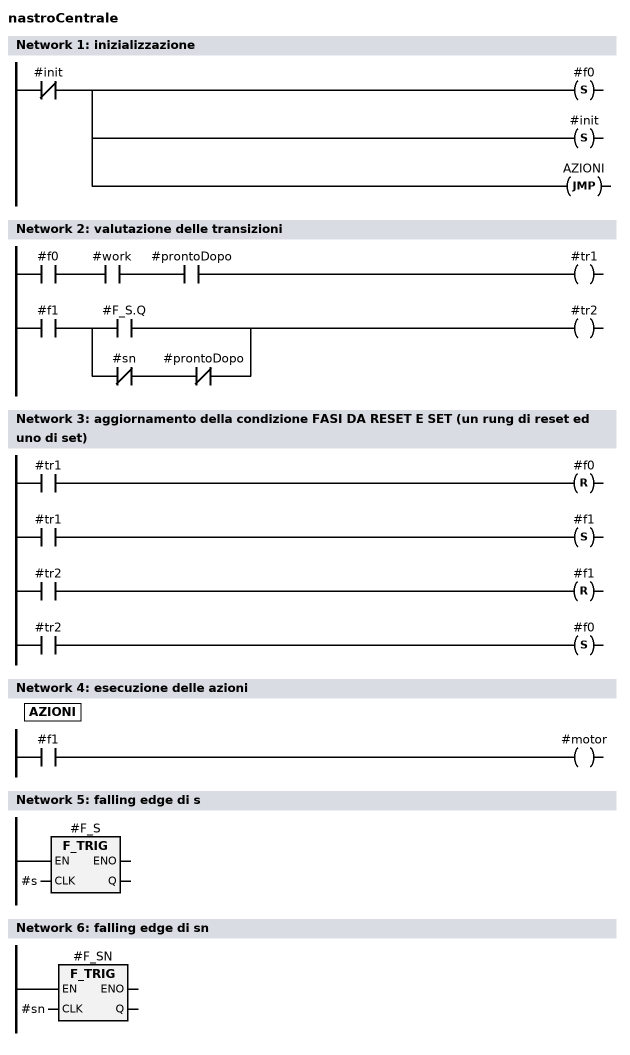
   RUNG wire#powerrail
      I_Contact( #init )
      wire#w1
      S_Coil( #f0 )
   END_RUNG
   RUNG wire#w1
      S_Coil( #init )
   END_RUNG
   RUNG wire#w1
      JumpCoil( AZIONI )
   END_RUNG
   // the same network as SCL:
   IF NOT #init THEN #f0 := TRUE; END_IF;
   #_w1 := NOT #init;
   IF #_w1 THEN
       #init := TRUE;
       GOTO AZIONI;
   END_IF;
END_REGION

REGION Network 2: valutazione delle transizioni
   RUNG wire#powerrail
      Contact( #f0 )
      Contact( #work )
      Contact( #prontoDopo )
      Coil( #tr1 )
   END_RUNG
   RUNG wire#powerrail
      Contact( #f1 )
      wire#w1
      Contact( #F_S.Q )
      wire#w2
      Coil( #tr2 )
   END_RUNG
   RUNG wire#w1
      I_Contact( #sn )
      I_Contact( #prontoDopo )
   END_RUNG wire#w2
   // the same network as SCL:
   #tr1 := #f0 AND #work AND #prontoDopo;
   #tr2 := #f1 AND (#F_S.Q OR (NOT #sn AND NOT #prontoDopo));
END_REGION

REGION Network 3: aggiornamento della condizione FASI DA RESET E SET (un rung di reset ed uno di set)
   RUNG wire#powerrail
      Contact( #tr1 )
      R_Coil( #f0 )
   END_RUNG
   RUNG wire#powerrail
      Contact( #tr1 )
      S_Coil( #f1 )
   END_RUNG
   RUNG wire#powerrail
      Contact( #tr2 )
      R_Coil( #f1 )
   END_RUNG
   RUNG wire#powerrail
      Contact( #tr2 )
      S_Coil( #f0 )
   END_RUNG
   // the same network as SCL:
   IF #tr1 THEN
       #f0 := FALSE;
       #f1 := TRUE;
   END_IF;
   IF #tr2 THEN
       #f1 := FALSE;
       #f0 := TRUE;
   END_IF;
END_REGION

REGION Network 4: esecuzione delle azioni
   Label( AZIONI )
   RUNG wire#powerrail
      Contact( #f1 )
      Coil( #motor )
   END_RUNG
   // the same network as SCL:
   AZIONI:
   #motor := #f1;
END_REGION

REGION Network 5: falling edge di s
   #F_S(CLK := #s);   // F_TRIG
END_REGION

REGION Network 6: falling edge di sn
   #F_SN(CLK := #sn);   // F_TRIG
END_REGION
END_FUNCTION_BLOCK

FUNCTION_BLOCK "NastroDirezionale"   // FB7, LAD
{ S7_Optimized_Access := 'TRUE' }
VERSION : 0.1
   VAR_INPUT
      visionSens : Bool;
      Sdestro : Bool;   // sensore del nastro Destro (conferma dello spostamento a destra del pacco)
      BoxOn : Bool;
      prontoDopo : Bool;
   END_VAR
   VAR_OUTPUT
      motor : Bool;
      nastroDestra : Bool;
      work_finished : Bool;
   END_VAR
   VAR
      init : Bool;
      f0 : Bool;
      f1 : Bool;
      f2 : Bool;
      F_S : F_TRIG;
      R_BoxOn : R_TRIG;
   END_VAR
   VAR_TEMP
      tr1 : Bool;
      tr2 : Bool;
      tr3 : Bool;
   END_VAR
   VAR_TEMP   // added for the SCL form of the ladder/FBD networks
      _w1 : Bool;
   END_VAR
BEGIN

REGION Network 1: inizializzazione
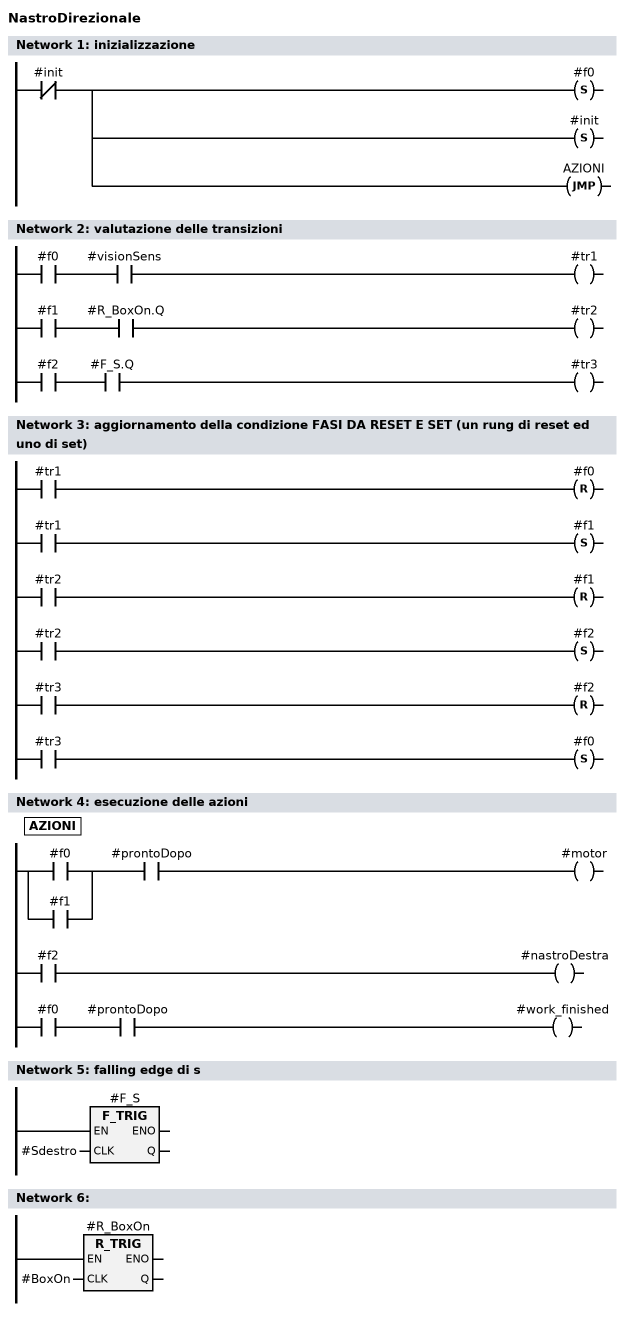
   RUNG wire#powerrail
      I_Contact( #init )
      wire#w1
      S_Coil( #f0 )
   END_RUNG
   RUNG wire#w1
      S_Coil( #init )
   END_RUNG
   RUNG wire#w1
      JumpCoil( AZIONI )
   END_RUNG
   // the same network as SCL:
   IF NOT #init THEN #f0 := TRUE; END_IF;
   #_w1 := NOT #init;
   IF #_w1 THEN
       #init := TRUE;
       GOTO AZIONI;
   END_IF;
END_REGION

REGION Network 2: valutazione delle transizioni
   RUNG wire#powerrail
      Contact( #f0 )
      Contact( #visionSens )
      Coil( #tr1 )
   END_RUNG
   RUNG wire#powerrail
      Contact( #f1 )
      Contact( #R_BoxOn.Q )
      Coil( #tr2 )
   END_RUNG
   RUNG wire#powerrail
      Contact( #f2 )
      Contact( #F_S.Q )
      Coil( #tr3 )
   END_RUNG
   // the same network as SCL:
   #tr1 := #f0 AND #visionSens;
   #tr2 := #f1 AND #R_BoxOn.Q;
   #tr3 := #f2 AND #F_S.Q;
END_REGION

REGION Network 3: aggiornamento della condizione FASI DA RESET E SET (un rung di reset ed uno di set)
   RUNG wire#powerrail
      Contact( #tr1 )
      R_Coil( #f0 )
   END_RUNG
   RUNG wire#powerrail
      Contact( #tr1 )
      S_Coil( #f1 )
   END_RUNG
   RUNG wire#powerrail
      Contact( #tr2 )
      R_Coil( #f1 )
   END_RUNG
   RUNG wire#powerrail
      Contact( #tr2 )
      S_Coil( #f2 )
   END_RUNG
   RUNG wire#powerrail
      Contact( #tr3 )
      R_Coil( #f2 )
   END_RUNG
   RUNG wire#powerrail
      Contact( #tr3 )
      S_Coil( #f0 )
   END_RUNG
   // the same network as SCL:
   IF #tr1 THEN
       #f0 := FALSE;
       #f1 := TRUE;
   END_IF;
   IF #tr2 THEN
       #f1 := FALSE;
       #f2 := TRUE;
   END_IF;
   IF #tr3 THEN
       #f2 := FALSE;
       #f0 := TRUE;
   END_IF;
END_REGION

REGION Network 4: esecuzione delle azioni
   Label( AZIONI )
   RUNG wire#powerrail
      Contact( #f0 )
      wire#w1
      Contact( #prontoDopo )
      Coil( #motor )
   END_RUNG
   RUNG wire#powerrail
      Contact( #f1 )
   END_RUNG wire#w1
   RUNG wire#powerrail
      Contact( #f2 )
      Coil( #nastroDestra )
   END_RUNG
   RUNG wire#powerrail
      Contact( #f0 )
      Contact( #prontoDopo )
      Coil( #work_finished )
   END_RUNG
   // the same network as SCL:
   AZIONI:
   #motor := (#f0 OR #f1) AND #prontoDopo;
   #nastroDestra := #f2;
   #work_finished := #f0 AND #prontoDopo;
END_REGION

REGION Network 5: falling edge di s
   #F_S(CLK := #Sdestro);   // F_TRIG
END_REGION

REGION Network 6
   #R_BoxOn(CLK := #BoxOn);   // R_TRIG
END_REGION
END_FUNCTION_BLOCK

FUNCTION "MHJ-PLC-Lab-Function-S71200" : Void   // FC9000, SCL
{ S7_Optimized_Access := 'TRUE' }
VERSION : 0.1
   VAR_TEMP
      rdTimeReturn : Int;
      outputTime : DTL;
      SyncVal : Byte;
      forVal : Int;
      forVal_2 : Int;
      Value : Byte;
   END_VAR
   VAR CONSTANT
      CompVal : Byte := 16#34;
      Value_01 : Byte := 16#11;
      Value_01_DW : DWord := 16#A165_D992;
      Value_02_DW : DWord := 16#58BE_4401;
   END_VAR
BEGIN

   #Value:=PEEK(area := 16#82,
        dbNumber := 0,
        byteOffset := 511);
   #Value := #Value + 1;

   POKE(area := 16#82,
        dbNumber := 0,
        byteOffset := 511,
        value := #Value);

   POKE(area:=16#81,
        dbNumber:=0,
        byteOffset:=1016,
        value:=#Value_01_DW);
   POKE(area := 16#81,
        dbNumber := 0,
        byteOffset := 1020,
        value := #Value_02_DW);

   POKE(area := 16#81,
        dbNumber := 0,
        byteOffset := 511,
        value := B#16#00);

   FOR #forVal := 0 TO 120 DO
       FOR #forVal_2:=0 TO 10 DO
           #rdTimeReturn:=RD_SYS_T(#outputTime);
           #rdTimeReturn := WR_SYS_T(#outputTime);
           #rdTimeReturn := RD_SYS_T(#outputTime);
           #rdTimeReturn := WR_SYS_T(#outputTime);
       END_FOR;
       #SyncVal:= PEEK(area := 16#81,
                      dbNumber := 0,
                      byteOffset := 511);
       IF #SyncVal = #CompVal THEN
          GOTO M_1;
       END_IF;
   END_FOR;
   RETURN;

   M_1:
   POKE(area := 16#81,
        dbNumber := 0,
        byteOffset := 511,
        value := B#16#0);
END_FUNCTION

ORGANIZATION_BLOCK "Main"   // OB1, LAD, ProgramCycle
TITLE = "Main Program Sweep (Cycle)"
{ S7_Optimized_Access := 'TRUE' }
VERSION : 0.1
   VAR_INPUT
      Initial_Call : Bool;   // Initial call of this OB
      Remanence : Bool;   // =True, if remanent data are available
   END_VAR
   VAR_TEMP
      Tag_24 : Bool;
      Tag_25 : Real;
   END_VAR
   VAR_TEMP   // added for the SCL form of the ladder/FBD networks
      _w1 : Bool;
   END_VAR
BEGIN

REGION Network 1: Konnektierungsbaustein für PLC-Lab
   // Im Netzwerk 1 wird der Konnektierungsbaustein für PLC-Lab aufgerufen.
   // Dieser Aufruf darf nicht entfernt werden!
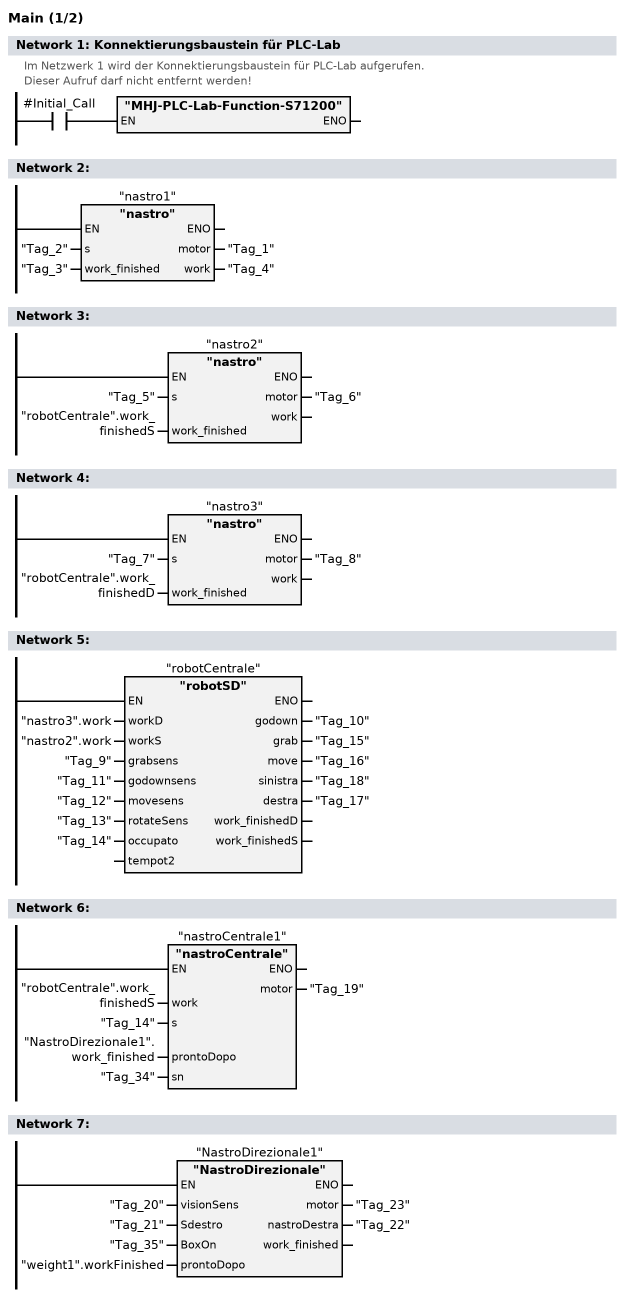
   RUNG wire#powerrail
      Contact( #Initial_Call )
      "MHJ-PLC-Lab-Function-S71200"()
   END_RUNG
   // the same network as SCL:
   IF #Initial_Call THEN "MHJ-PLC-Lab-Function-S71200"(); END_IF;
END_REGION

REGION Network 2
   RUNG wire#powerrail
      "nastro1"(s := "Tag_2", work_finished := "Tag_3", motor => "Tag_1", work => "Tag_4")
   END_RUNG
   // the same network as SCL:
   "nastro1"(s := "Tag_2", work_finished := "Tag_3", motor => "Tag_1", work => "Tag_4");   // "nastro"
END_REGION

REGION Network 3
   RUNG wire#powerrail
      "nastro2"(s := "Tag_5", work_finished := "robotCentrale".work_finishedS, motor => "Tag_6", work =>)
   END_RUNG
   // the same network as SCL:
   "nastro2"(s := "Tag_5", work_finished := "robotCentrale".work_finishedS, motor => "Tag_6");   // "nastro"
END_REGION

REGION Network 4
   RUNG wire#powerrail
      "nastro3"(s := "Tag_7", work_finished := "robotCentrale".work_finishedD, motor => "Tag_8", work =>)
   END_RUNG
   // the same network as SCL:
   "nastro3"(s := "Tag_7", work_finished := "robotCentrale".work_finishedD, motor => "Tag_8");   // "nastro"
END_REGION

REGION Network 5
   RUNG wire#powerrail
      "robotCentrale"(workD := "nastro3".work, workS := "nastro2".work, grabsens := "Tag_9", godownsens := "Tag_11", movesens := "Tag_12", rotateSens := "Tag_13", occupato := "Tag_14", tempot2 :=, godown => "Tag_10", grab => "Tag_15", move => "Tag_16", sinistra => "Tag_18", destra => "Tag_17", work_finishedD =>, work_finishedS =>)
   END_RUNG
   // the same network as SCL:
   "robotCentrale"(workD := "nastro3".work,   // "robotSD"
                   workS := "nastro2".work,
                   grabsens := "Tag_9",
                   godownsens := "Tag_11",
                   movesens := "Tag_12",
                   rotateSens := "Tag_13",
                   occupato := "Tag_14",
                   godown => "Tag_10",
                   grab => "Tag_15",
                   move => "Tag_16",
                   sinistra => "Tag_18",
                   destra => "Tag_17");
END_REGION

REGION Network 6
   RUNG wire#powerrail
      "nastroCentrale1"(work := "robotCentrale".work_finishedS, s := "Tag_14", prontoDopo := "NastroDirezionale1".work_finished, sn := "Tag_34", motor => "Tag_19")
   END_RUNG
   // the same network as SCL:
   "nastroCentrale1"(work := "robotCentrale".work_finishedS,   // "nastroCentrale"
                     s := "Tag_14",
                     prontoDopo := "NastroDirezionale1".work_finished,
                     sn := "Tag_34",
                     motor => "Tag_19");
END_REGION

REGION Network 7
   RUNG wire#powerrail
      "NastroDirezionale1"(visionSens := "Tag_20", Sdestro := "Tag_21", BoxOn := "Tag_35", prontoDopo := "weight1".workFinished, motor => "Tag_23", nastroDestra => "Tag_22", work_finished =>)
   END_RUNG
   // the same network as SCL:
   "NastroDirezionale1"(visionSens := "Tag_20",   // "NastroDirezionale"
                        Sdestro := "Tag_21",
                        BoxOn := "Tag_35",
                        prontoDopo := "weight1".workFinished,
                        motor => "Tag_23",
                        nastroDestra => "Tag_22");
END_REGION

REGION Network 8
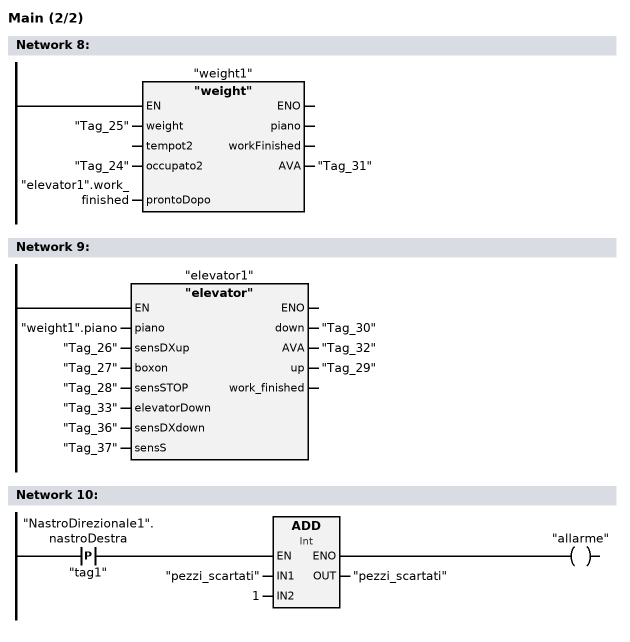
   RUNG wire#powerrail
      "weight1"(weight := "Tag_25", tempot2 :=, occupato2 := "Tag_24", prontoDopo := "elevator1".work_finished, piano =>, workFinished =>, AVA => "Tag_31")
   END_RUNG
   // the same network as SCL:
   "weight1"(weight := "Tag_25",   // "weight"
             occupato2 := "Tag_24",
             prontoDopo := "elevator1".work_finished,
             AVA => "Tag_31");
END_REGION

REGION Network 9
   RUNG wire#powerrail
      "elevator1"(piano := "weight1".piano, sensDXup := "Tag_26", boxon := "Tag_27", sensSTOP := "Tag_28", elevatorDown := "Tag_33", sensDXdown := "Tag_36", sensS := "Tag_37", down => "Tag_30", AVA => "Tag_32", up => "Tag_29", work_finished =>)
   END_RUNG
   // the same network as SCL:
   "elevator1"(piano := "weight1".piano,   // "elevator"
               sensDXup := "Tag_26",
               boxon := "Tag_27",
               sensSTOP := "Tag_28",
               elevatorDown := "Tag_33",
               sensDXdown := "Tag_36",
               sensS := "Tag_37",
               down => "Tag_30",
               AVA => "Tag_32",
               up => "Tag_29");
END_REGION

REGION Network 10
   RUNG wire#powerrail
      P_Contact(operand := "NastroDirezionale1".nastroDestra, bit := "tag1")
      { S7_Templates := "SrcType := Int" } Add(in1 := "pezzi_scartati", in2 := 1, out => "pezzi_scartati")
      Coil( "allarme" )
   END_RUNG
   // the same network as SCL:
   #_w1 := "NastroDirezionale1".nastroDestra AND NOT "tag1";   // rising edge of "NastroDirezionale1".nastroDestra
   "tag1" := "NastroDirezionale1".nastroDestra;
   IF #_w1 THEN "pezzi_scartati" := "pezzi_scartati" + 1; END_IF;
   "allarme" := #_w1;
END_REGION
END_ORGANIZATION_BLOCK

(* ===== HMI "HMI_RT_1" =====
system functions are stored by id; their names below are inferred from use
connection "HMI_Connection_1": ETHERNET, SMART_S7_1200_OMS

HMI tags "Default tag table"
   "Tag_ScreenNumber" : UInt, internal
   "pezzi_scartati" : Int = PLC pezzi_scartati AT %MW0, 1 s

analog alarms
   1: '', class Errors, trigger "pezzi_scartati"

Template "Template_1" 800x480
   Button "Exit" at 722,440 size 55x39; TextOff 'Exit'; PictureOff "ExitRuntime_KTP900_Basic_PN_TR"; PictureOn "ExitRuntime_KTP900_Basic_PN_TR"
      on Release: StopRuntime(0)
   Button "Template_Button" at 622,440 size 55x39; TextOff 'Text'
   Button "Template_Button_1" at 522,440 size 55x39; TextOff 'Text'
   Button "Template_Button_2" at 422,440 size 55x39; TextOff 'Text'
   Button "Template_Button_3" at 322,440 size 55x39; TextOff 'Text'
   Button "Template_Button_4" at 222,440 size 55x39; TextOff 'Text'
   Button "Alarms" at 122,440 size 55x39; TextOff 'Alarms'; PictureOff "AlarmDisplay_KTP900_Basic_PN_TR"; PictureOn "AlarmDisplay_KTP900_Basic_PN_TR"
      on Release: function_ef3f5d25("Alarm window_Unacknowledged", -1)
   Button "Start screen" at 22,440 size 55x39; TextOff 'Start screen'; PictureOff "NavigateHome_KTP900_Basic_PN_TR"; PictureOn "NavigateHome_KTP900_Basic_PN_TR"
      on Release: ActivateScreen("Root screen", 0)
   SymbolicIOField "Symbolic_IO_Field_Screen" at 73,7 size 620x26; TextOff '0'; TextOn '1'; TextList "TextList_ScreenNames"
      ProcessValue <- "Tag_ScreenNumber"
      on Change: ActivateScreenByNumber("Tag_ScreenNumber", 0)
   DateTimeField "HmiScreenItemData" at 695,20 size 105x20
   DateTimeField "HmiScreenItemData_1" at 695,0 size 105x20
   GraphicView "Logo" at 0,0 size 71x40; Picture "Logo of HMI_1"

screen "Root screen" 800x480, template "Template_1"
   on GenerateScreen: SetTag("Tag_ScreenNumber", 1)
   TextField "HmiScreenItemData" at 76,198 size 640x22; Text 'ALLARME TROPPI SCARTI IN MAGAZZINO'
   Circle "Circle_1" at 354,125 size 73x73
      Appearance <- "pezzi_scartati"
   IOField "I/O field_1" at 354,293 size 96x32; FormatPattern s99
      ProcessValue <- "pezzi_scartati"
*)